// TIA Portal project "InfocomTIALibV16" (V16)

(* hardware
DEVICE "S7-1200 station_1"  S7-1200 Station
   slot 0: "Rack_0"  S7-1200 Rack  Rack  V1.0
   slot 1: "PLC_1"  CPU 1217C DC/DC/DC  6ES7 217-1AG40-0XB0  V4.4
DEVICE "S7300/ET200M station_1"  S7-300 station
   slot 0: "Rail_0"  Rail  6ES7 390-1***0-0AA0
   slot 2: "PLC_2"  CPU 315-2 PN/DP  6ES7 315-2EH14-0AB0  V3.2
      slot 2: "PROFINET interface_1"  PN-IO
         slot 1: "Port_1"  Port
         slot 2: "Port_2"  Port
*)

// ===== PLC "PLC_1"  CPU 1217C DC/DC/DC =====

FUNCTION_BLOCK "TimeS"   // FB2, SCL
{ S7_Optimized_Access := 'TRUE' }
VERSION : 0.1
   VAR_INPUT
      IN : Bool;
      PT : Int := 1;   // (0 < PT < 3600)
      Mode : Int := 2;   // 0=Pulse, 1=ExtP, 2=OnDel, 3=RetOn, 4=OffDel
      Reset : Bool;
   END_VAR
   VAR_OUTPUT
      OUT : Bool;
      InvOUT : Bool;
   END_VAR
   VAR
      DTL_NOW : DTL;
      DTL_FINISH : DTL;
      front : Bool;
      PT_Time : Time;
   END_VAR
   VAR_TEMP
      statusWord : Int;
      tPT : Int;
   END_VAR
   VAR CONSTANT
      MS_IN_1S : Int := 1000;
      SEC_IN_1MM : Int := 60;
   END_VAR
BEGIN
   #statusWord := RD_SYS_T(#DTL_NOW);//Read system time.
   #tPT := LIMIT(MN := 0, IN := #PT, MX := 3600);
   IF NOT #front AND #IN THEN
       #PT_Time := DINT_TO_TIME(INT_TO_DINT(#PT) * #MS_IN_1S); //Convert PT to time.
       #DTL_FINISH := T_ADD(IN1 := #DTL_NOW, IN2 := #PT_Time);//Calculate Finish time.
       #front := true;//Front was detected.
   END_IF;
   IF NOT #IN THEN
       #front := false;
   END_IF;

   CASE #Mode OF
           //----------------------------------------------------------------------------------------
       0:  //0=Pulse, Пуск таймера в виде импульса
           IF #IN AND #DTL_NOW <= #DTL_FINISH AND NOT #Reset THEN
               #OUT := TRUE;
           ELSE
               #OUT := FALSE;
           END_IF;
           //----------------------------------------------------------------------------------------
       1:  //1=ExtP,Пуск таймера в виде импульса с увеличенной длительностью
           IF #DTL_NOW <= #DTL_FINISH THEN
               #OUT := TRUE;
           ELSE
               #OUT := FALSE;
           END_IF;
           //----------------------------------------------------------------------------------------
       2:  //2=OnDel, Пуск таймера с задержкой включения
           IF #IN AND #DTL_NOW >= #DTL_FINISH AND NOT #Reset THEN
               #OUT := true;
           ELSE
               #OUT := false;
           END_IF;
           //----------------------------------------------------------------------------------------
       3:  //3=RetOn, Пуск таймера с задержкой включения с функцией накопления
           IF TRUE THEN
               ;
           ELSE
               ;
           END_IF;
           //----------------------------------------------------------------------------------------
       4:  //4=OffDel, Пуск таймера с задержкой выключения
           IF TRUE THEN
               ;
           ELSE
               ;
           END_IF;
           //----------------------------------------------------------------------------------------
       ELSE  //Out = FALSE
           #OUT := FALSE;

   END_CASE;
END_FUNCTION_BLOCK

ORGANIZATION_BLOCK "Main"   // OB1, LAD, ProgramCycle
TITLE = "Main Program Sweep (Cycle)"
{ S7_Optimized_Access := 'TRUE' }
VERSION : 0.1
   VAR_INPUT
      Initial_Call : Bool;   // Initial call of this OB
      Remanence : Bool;   // =True, if remanent data are available
   END_VAR
BEGIN
END_ORGANIZATION_BLOCK

// ===== PLC "PLC_2"  CPU 315-2 PN/DP =====

DATA_BLOCK "TimerS_DB"   // DB1
{ S7_Optimized_Access := 'FALSE' }
VERSION : 0.1
// stored: InstanceOfName TimerS
"TimerS"
BEGIN
END_DATA_BLOCK

FUNCTION_BLOCK "TimerS"   // FB1, SCL
{ S7_Optimized_Access := 'FALSE' }
VERSION : 0.1
   VAR_INPUT
      IN : Bool;
      PT : Int;   // (0 < PT < 3600)
      Mode : Int;   // 0=Pulse, 1=ExtP, 2=OnDel, 3=RetOn, 4=OffDel (Def val = 0)
      Reset : Bool;
   END_VAR
   VAR_OUTPUT
      OUT : Bool;
      InvOUT : Bool;
   END_VAR
   VAR
      DTL_NOW : Date_And_Time;
      DTL_FINISH : Date_And_Time;
      PT_Time : Time;
      FP_IN : "Front";   // Front
      FN_IN : "Front";   // Front
   END_VAR
   VAR_TEMP
      statusWord : Int;
      tPT : Int;
      tMode : Int;
   END_VAR
   VAR CONSTANT
      MS_IN_1S : Int := 1000;
   END_VAR
BEGIN
   #statusWord := RD_SYS_T(#DTL_NOW);//Read system time.
   #tPT := LIMIT(MN := 0, IN := #PT, MX := 3600);//Check input param
   #tMode := LIMIT(MN := 0, IN := #Mode, MX := 4);
   #FP_IN(IN:=#IN);
   #FN_IN(IN := NOT #IN);

   IF #FP_IN.OUT THEN
       #PT_Time := DINT_TO_TIME(INT_TO_DINT(#tPT) * #MS_IN_1S); //Convert PT to time.
       #DTL_FINISH := T_ADD(IN1 := #DTL_NOW, IN2 := #PT_Time);//Calculate Finish time.
   END_IF;


   CASE #tMode OF
           //----------------------------------------------------------------------------------------
       0:  //0=Pulse, Пуск таймера в виде импульса
           IF #FP_IN.OUT THEN
               #PT_Time := DINT_TO_TIME(INT_TO_DINT(#tPT) * #MS_IN_1S); //Convert PT to time.
               #DTL_FINISH := T_ADD(IN1 := #DTL_NOW, IN2 := #PT_Time);//Calculate Finish time.
           END_IF;
           IF #IN AND #DTL_NOW T_COMP #DTL_FINISH AND NOT #Reset THEN
               #OUT := TRUE;
           END_IF;
           IF NOT #IN OR #DTL_NOW T_COMP #DTL_FINISH OR #Reset THEN
               #OUT := FALSE;
           END_IF;
           //----------------------------------------------------------------------------------------
       1:  //1=ExtP,Пуск таймера в виде импульса с увеличенной длительностью
           IF #FP_IN.OUT THEN
               #PT_Time := DINT_TO_TIME(INT_TO_DINT(#tPT) * #MS_IN_1S); //Convert PT to time.
               #DTL_FINISH := T_ADD(IN1 := #DTL_NOW, IN2 := #PT_Time);//Calculate Finish time.
           END_IF;
           IF #DTL_NOW T_COMP #DTL_FINISH THEN
               #OUT := TRUE;
           ELSE
               #OUT := FALSE;
           END_IF;
           //----------------------------------------------------------------------------------------
       2:  //2=OnDel, Пуск таймера с задержкой включения
           IF #FP_IN.OUT THEN
               #PT_Time := DINT_TO_TIME(INT_TO_DINT(#tPT) * #MS_IN_1S); //Convert PT to time.
               #DTL_FINISH := T_ADD(IN1 := #DTL_NOW, IN2 := #PT_Time);//Calculate Finish time.
           END_IF;
           IF #IN AND #DTL_NOW T_COMP #DTL_FINISH AND NOT #Reset THEN
               #OUT := true;
           END_IF;
           IF NOT #IN  OR #Reset OR #DTL_NOW T_COMP #DTL_FINISH THEN
               #OUT := false;
           END_IF;
           //----------------------------------------------------------------------------------------
       3:  //3=RetOn, Пуск таймера с задержкой включения с функцией накопления
           IF #FP_IN.OUT THEN
               #PT_Time := DINT_TO_TIME(INT_TO_DINT(#tPT) * #MS_IN_1S); //Convert PT to time.
               #DTL_FINISH := T_ADD(IN1 := #DTL_NOW, IN2 := #PT_Time);//Calculate Finish time.
           END_IF;
           IF #IN AND #DTL_NOW T_COMP #DTL_FINISH THEN
               #OUT := true;
           END_IF;
           IF #Reset THEN
               #OUT := FALSE;
           END_IF;
           //----------------------------------------------------------------------------------------
       4:  //4=OffDel, Пуск таймера с задержкой выключения
           IF #FN_IN.OUT THEN
               #PT_Time := DINT_TO_TIME(INT_TO_DINT(#tPT) * #MS_IN_1S); //Convert PT to time.
               #DTL_FINISH := T_ADD(IN1 := #DTL_NOW, IN2 := #PT_Time);//Calculate Finish time.
           END_IF;
           IF #IN OR #DTL_NOW T_COMP #DTL_FINISH AND NOT #Reset THEN
               #OUT := true;
           END_IF;
           IF #DTL_NOW T_COMP #DTL_FINISH OR #Reset THEN
               #OUT := false;
           END_IF;
           //----------------------------------------------------------------------------------------
       ELSE  //Out = FALSE
           #OUT := FALSE;

   END_CASE;
END_FUNCTION_BLOCK

FUNCTION_BLOCK "Front"   // FB2, SCL
{ S7_Optimized_Access := 'FALSE' }
VERSION : 0.1
   VAR_INPUT
      IN : Bool;
   END_VAR
   VAR_OUTPUT
      OUT : Bool;
   END_VAR
   VAR
      MEMORY : Bool;
   END_VAR
BEGIN
   IF #IN AND NOT #MEMORY THEN
       #OUT := TRUE;
       #MEMORY := TRUE;
   ELSE
       #OUT := FALSE;
   END_IF;
   IF NOT #IN THEN
       #MEMORY := FALSE;
   END_IF;
END_FUNCTION_BLOCK

FUNCTION_BLOCK "Valve"   // FB3, SCL
{ S7_Optimized_Access := 'FALSE' }
VERSION : 0.1
   VAR_INPUT
      isModAuto : Bool;
      isModMan : Bool;
      isModLocal : Bool;
      cmdOpenAuto : Bool;
      cmdCloseAuto : Bool;
      cmdOpenLocal : Bool;
      cmdCloseLocal : Bool;
      isOpen : Bool;
      isClose : Bool;
      isPermit : Bool;
      isIntlock : Bool;
      isProtect : Bool;
      isFaultExt : Bool;
      cmdRst : Bool;
      MonTime : Int;
      ctrlWord : Word;
   END_VAR
   VAR_OUTPUT
      isGrpError : Bool;
      Ctrl : Bool;
      AutoAct : Bool;
      ManAct : Bool;
      LocalAct : Bool;
      RdyToStart : Bool;
      RdyToReset : Bool;
   END_VAR
   VAR
      isFault : Bool;
      TOpening : "TimerS";
      isLocked : Bool;
   END_VAR
BEGIN
   #AutoAct := #isModAuto AND NOT #isModMan AND NOT #isModLocal;
   #ManAct := #isModMan AND NOT #isModLocal;
   #LocalAct := #isModLocal;

   IF #cmdRst THEN
       #isFault := false;
   END_IF;

   IF #isClose AND #isOpen THEN
       #isFault := TRUE;
   END_IF;

   IF (#cmdOpenAuto  AND #cmdCloseAuto) OR (#cmdOpenLocal AND  #cmdCloseLocal) THEN
       #isFault := TRUE;
   END_IF;

   #TOpening(IN:=#Ctrl AND NOT #isOpen,
             PT:=#MonTime,
             Mode:=2);

   IF #TOpening.OUT THEN
       #isFault := TRUE;
   END_IF;

   #isLocked := #isPermit OR #isIntlock OR #isProtect;
   IF #isLocked THEN
       #isFault := TRUE;
   END_IF;


   #isGrpError := #isFaultExt OR #isFault;

   #Ctrl := (#AutoAct AND #cmdOpenAuto AND NOT #cmdCloseAuto) OR (#LocalAct AND #cmdOpenLocal AND NOT #cmdCloseLocal) AND NOT #isLocked;
END_FUNCTION_BLOCK

ORGANIZATION_BLOCK "Main"   // OB1, LAD
TITLE = "Main Program Sweep (Cycle)"
{ S7_Optimized_Access := 'FALSE' }
VERSION : 0.1
   VAR_TEMP
      OB1_EV_CLASS : Byte;   // Bits 0-3 = 1 (Coming event), Bits 4-7 = 1 (Event class 1)
      OB1_SCAN_1 : Byte;   // 1 (Cold restart scan 1 of OB 1), 3 (Scan 2-n of OB 1)
      OB1_PRIORITY : Byte;   // Priority of OB Execution
      OB1_OB_NUMBR : Byte;   // 1 (Organization block 1, OB1)
      OB1_RESERVED_1 : Byte;   // Reserved for system
      OB1_RESERVED_2 : Byte;   // Reserved for system
      OB1_PREV_CYCLE : Int;   // Cycle time of previous OB1 scan (milliseconds)
      OB1_MIN_CYCLE : Int;   // Minimum cycle time of OB1 (milliseconds)
      OB1_MAX_CYCLE : Int;   // Maximum cycle time of OB1 (milliseconds)
      OB1_DATE_TIME : Date_And_Time;   // Date and time OB1 started
   END_VAR
BEGIN

REGION Network 1
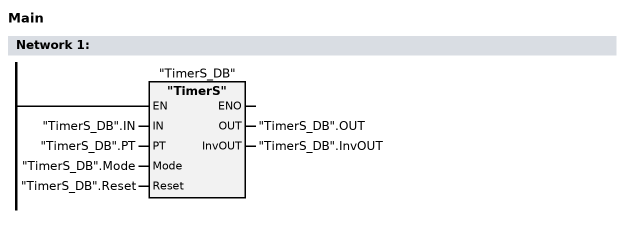
   RUNG wire#powerrail
      "TimerS_DB"(IN := "TimerS_DB".IN, PT := "TimerS_DB".PT, Mode := "TimerS_DB".Mode, Reset := "TimerS_DB".Reset, OUT => "TimerS_DB".OUT, InvOUT => "TimerS_DB".InvOUT)
   END_RUNG
   // the same network as SCL:
   "TimerS_DB"(IN := "TimerS_DB".IN,   // "TimerS"
               PT := "TimerS_DB".PT,
               Mode := "TimerS_DB".Mode,
               Reset := "TimerS_DB".Reset,
               OUT => "TimerS_DB".OUT,
               InvOUT => "TimerS_DB".InvOUT);
END_REGION
END_ORGANIZATION_BLOCK